// TIA Portal V19 export
FUNCTION "Prod_O_TODO_Swap" : Bool   // FC71, LAD
// stored: SetENOAutomatically false
   VAR_INPUT
      Index_A : Int;
      Index_B : Int;
   END_VAR
   VAR_TEMP
      OK : Bool;
      ItemCopy : "Prod_Item";
   END_VAR
BEGIN

REGION Network 1
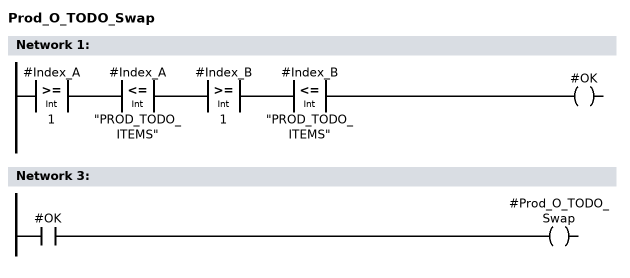
   RUNG wire#powerrail
      { S7_Templates := "SrcType := Int" } GE_Contact(in1 := #Index_A, in2 := 1)
      { S7_Templates := "SrcType := Int" } LE_Contact(in1 := #Index_A, in2 := "PROD_TODO_ITEMS")
      { S7_Templates := "SrcType := Int" } GE_Contact(in1 := #Index_B, in2 := 1)
      { S7_Templates := "SrcType := Int" } LE_Contact(in1 := #Index_B, in2 := "PROD_TODO_ITEMS")
      Coil( #OK )
   END_RUNG
   // the same network as SCL:
   #OK := (#Index_A >= 1) AND (#Index_A <= "PROD_TODO_ITEMS") AND (#Index_B >= 1) AND (#Index_B <= "PROD_TODO_ITEMS");
END_REGION

REGION Network 2 (SCL)
   IF #OK THEN
       #ItemCopy := "Production".O_TODO[#Index_A];
       "Production".O_TODO[#Index_A] := "Production".O_TODO[#Index_B];
       "Production".O_TODO[#Index_B] := #ItemCopy;
   END_IF;
END_REGION

REGION Network 3
   RUNG wire#powerrail
      Contact( #OK )
      Coil( #Prod_O_TODO_Swap )
   END_RUNG
   // the same network as SCL:
   #Prod_O_TODO_Swap := #OK;
END_REGION
END_FUNCTION
